FUNCTION_BLOCK fbRawRatioConversionAllenINV
VAR_INPUT

	iRawData : INT;
	rRawRatio : LREAL;


END_VAR
VAR_OUTPUT

	rConvertedResult : INT;
END_VAR
VAR
	rRawData: LREAL;
	rConvertedResult_1: LREAL;
END_VAR

rRawData := INT_TO_LREAL (iRawData);

IF rRawData <> 0 AND rRawRatio <> 0 THEN
rConvertedResult_1 := rRawData * rRawRatio;
END_IF

IF rRawData = 0 OR rRawRatio = 0 THEN
rConvertedResult := 0;
END_IF

rConvertedResult := LREAL_TO_INT(rConvertedResult_1);

END_FUNCTION_BLOCK

(* stored: Version 1.1.0.1, ProductVersion 3.1.4024.12
   POU fbRawRatioConversionAllenINV: Id {1e5d7f0a-5e1c-4874-8e33-ee3dc160e077}, SpecialFunc None *)
